Yaskawa INFORM job: FRONT_WELD_-90ST-2_5040.JBI

/JOB
//NAME FRONT_WELD_-90ST-2_5040
///FOLDERNAME 02-SKRZYNIE_JOBS
//POS
///NPOS 31,31,0,6,0,0
///TOOL 0
///POSTYPE PULSE
///PULSE
C00000=0,-52278,40443,0,6873,-1
C00001=0,-52278,40443,0,6873,-1
C00002=0,-42686,23640,-7425,-34877,-70985
C00003=-25126,-44577,-4813,-57071,-34461,-49771
C00004=-6017,-48449,-29001,-102269,-8383,-26407
C00005=-2863,-32693,-8619,-87056,-6043,-33280
C00006=-4454,-30346,-5727,-85632,-7073,-34122
C00007=-4317,-30353,-5736,-85607,-6986,-34119
C00008=10744,-30180,-6062,-81609,2638,-34445
C00009=18416,-29401,-5585,-81961,7622,-33475
C00010=22266,-28575,-5017,-81243,10128,-33418
C00011=29231,-27482,-4303,-80552,14661,-33033
C00012=43222,-23908,-1841,-78421,23835,-32652
C00013=50847,-28145,-10545,-73666,29314,-34422
C00014=73589,-4766,14825,-76336,20345,-43289
C00015=78028,4989,28502,-80926,26481,-43407
C00016=77875,4741,28212,-80907,26383,-43432
C00017=74793,1589,24842,-81120,24540,-43763
C00018=78046,2413,16367,-60611,36178,-62151
C00019=71568,-5136,9623,-61706,29824,-60553
C00020=59451,-12704,5834,-65832,18507,-57161
C00021=58678,-17366,4552,-88847,13968,-42180
C00022=-23545,-30165,-21390,-32579,21562,-60781
C00023=-43411,-19640,-10965,1347,18370,-78573
C00024=-47411,-15989,-3853,13245,14656,-84014
C00025=-53847,-17736,-12367,37910,33155,-82886
C00026=-27070,-28432,-20556,12901,23133,-67942
C00027=-24971,-35737,-30976,9397,24510,-66000
C00028=0,-42686,23640,-7425,-34877,-70985
C00029=0,-52278,40443,-5610,-49281,-72137
C00030=0,-52278,40443,0,6873,-1
BC00000=744958
BC00001=774759
BC00002=903040
BC00003=940675
BC00004=971500
BC00005=971500
BC00006=971503
BC00007=971503
BC00008=971502
BC00009=971501
BC00010=971501
BC00011=971501
BC00012=971501
BC00013=971501
BC00014=971502
BC00015=971502
BC00016=971502
BC00017=971500
BC00018=971502
BC00019=971502
BC00020=971502
BC00021=971502
BC00022=971502
BC00023=971501
BC00024=971501
BC00025=971499
BC00026=971501
BC00027=971501
BC00028=903040
BC00029=774759
BC00030=774759
///POSTYPE BASE
///RECTAN
///RCONF 1,0,0,0,0,0,0,0,0,0,0,0,0,0,0,0,0,0,0,0,0,0,0,0
P00500=2.332,-5.281,-1.258,0.0000,0.0000,0.0000
///RCONF 0,0,0,0,0,0,0,0,0,0,0,0,0,0,0,0,0,0,0,0,0,0,0,0
P00501=-2.026,0.009,3.534,0.0000,0.0000,0.0000
///RCONF 1,0,0,0,0,0,0,0,0,0,0,0,0,0,0,0,0,0,0,0,0,0,0,0
P00502=-2.023,0.001,1.732,0.0000,0.0000,0.0000
P00503=0.138,-0.044,1.539,0.0000,0.0000,0.0000
P00504=-0.309,-0.010,1.636,0.0000,0.0000,0.0000
P00505=0.999,-9.916,8.214,0.0000,0.0000,0.0000
//INST
///DATE 2024/05/16 21:26
///ATTR SC,RW
///GROUP1 RB1,BS1
NOP
MOVJ C00000 BC00000 VJ=60.00
MOVJ C00001 BC00001 VJ=60.00
MOVJ C00002 BC00002 VJ=60.00
MOVJ C00003 BC00003 VJ=60.00
MOVJ C00004 BC00004 VJ=30.00
'::::::::::::::::::::::::::::::::
'W20
'::::::::::::::::::::::::::::::::
MOVL C00005 BC00005 V=333.3
SFTON P0503
MACRO1 MJ#(0) ARGF9
MOVL C00006 BC00006 V=166.7 PL=0
ARCON
MOVC C00007 BC00007 V=10.8
MOVC C00008 BC00008 V=10.8
MOVC C00009 BC00009 V=10.8
SFTOF
SFTON P0502
MOVC C00010 BC00010 V=10.8
MOVC C00011 BC00011 V=10.8
MOVC C00012 BC00012 V=10.8
ARCOF
MOVL C00013 BC00013 V=250.0
SFTOF
'::::::::::::::::::::::::::::::::
'W21
'::::::::::::::::::::::::::::::::
MOVL C00014 BC00014 V=666.7
SFTON P0500
MACRO1 MJ#(0) ARGF14
MOVL C00015 BC00015 V=166.7 PL=0
ARCON
MOVC C00016 BC00016 V=10.0
MOVC C00017 BC00017 V=10.0
MOVC C00018 BC00018 V=10.0
SFTOF
SFTON P0501
MOVC C00019 BC00019 V=10.0
MOVC C00020 BC00020 V=10.0
ARCOF
MOVL C00021 BC00021 V=166.7
SFTOF
MOVL C00022 BC00022 V=666.7
'::::::::::::::::::::::::::::::::
'W22
'::::::::::::::::::::::::::::::::
MOVL C00023 BC00023 V=333.3
SFTON P0505
MACRO1 MJ#(0) ARGF9
MOVL C00024 BC00024 V=166.7 PL=0
ARCON
MOVL C00025 BC00025 V=11.7
SFTOF
SFTON P0504
MOVL C00026 BC00026 V=11.7
ARCOF
MOVL C00027 BC00027 V=250.0
SFTOF
MOVJ C00028 BC00028 VJ=50.00
MOVJ C00029 BC00029 VJ=80.00
MOVJ C00030 BC00030 VJ=80.00
END
